// Mitsubishi GX Works2 project: BookEX2_3 Calculator   PLC: Q13UDV

// global labels: Global
VAR_GLOBAL
  bVar0 AT M5000 : BOOL;
  abArray0 AT M5010 : ARRAY [0..49] OF BOOL;
  sStr0 AT D5000 : STRING[199];
  sStr1 AT D5100 : STRING[199];
  sStr2 AT D5200 : STRING[199];
  sStr3 AT D5300 : STRING[199];
  sStr4 AT D5400 : STRING[199];
  sStr5 AT D5500 : STRING[199];
  sStr6 AT D5600 : STRING[199];
  sStr7 AT D5700 : STRING[199];
  sStr8 AT D5800 : STRING[199];
  sStr9 AT D5900 : STRING[199];
  iVar0 AT D4500 : INT;
  iVar1 AT D4501 : INT;
  iVar2 AT D4502 : INT;
  iVar3 AT D4503 : INT;
  iVar4 AT D4504 : INT;
  iVar5 AT D4505 : INT;
  iVar6 AT D4506 : INT;
  iVar7 AT D4507 : INT;
  iVar8 AT D4508 : INT;
  iVar9 AT D4509 : INT;
  dVar0 AT D4510 : DINT;
  dVar1 AT D4512 : DINT;
  dVar2 AT D4514 : DINT;
  dVar3 AT D4516 : DINT;
  dVar4 AT D4518 : DINT;
  dVar5 AT D4520 : DINT;
  dVar6 AT D4522 : DINT;
  dVar7 AT D4524 : DINT;
  dVar8 AT D4526 : DINT;
  dVar9 AT D4528 : DINT;
  wVar0 AT D4530 : WORD;
  wVar1 AT D4531 : WORD;
  wVar2 AT D4532 : WORD;
  wVar3 AT D4533 : WORD;
  wVar4 AT D4534 : WORD;
  wVar5 AT D4535 : WORD;
  wVar6 AT D4536 : WORD;
  wVar7 AT D4537 : WORD;
  wVar8 AT D4538 : WORD;
  wVar9 AT D4539 : WORD;
  dwVar0 AT D4540 : DWORD;
  dwVar1 AT D4542 : DWORD;
  dwVar2 AT D4544 : DWORD;
  dwVar3 AT D4546 : DWORD;
  dwVar4 AT D4548 : DWORD;
  dwVar5 AT D4550 : DWORD;
  dwVar6 AT D4552 : DWORD;
  dwVar7 AT D4554 : DWORD;
  dwVar8 AT D4556 : DWORD;
  dwVar9 AT D4558 : DWORD;
  fsVar0 AT D4560 : REAL;
  fsVar1 AT D4562 : REAL;
  fsVar2 AT D4564 : REAL;
  fsVar3 AT D4566 : REAL;
  fsVar4 AT D4568 : REAL;
  fsVar5 AT D4570 : REAL;
  fsVar6 AT D4572 : REAL;
  fsVar7 AT D4574 : REAL;
  fsVar8 AT D4576 : REAL;
  fsVar9 AT D4578 : REAL;
  fdVar0 AT D4580 : LREAL;
  tTime0 AT D4620 : TIME;
  tTime1 AT D4622 : TIME;
  tTime2 AT D4624 : TIME;
  tTime3 AT D4626 : TIME;
  tTime4 AT D4628 : TIME;
  tTime5 AT D4630 : TIME;
  tTime6 AT D4632 : TIME;
  tTime7 AT D4634 : TIME;
  tTime8 AT D4636 : TIME;
  tTime9 AT D4638 : TIME;
  tTime10 AT D4640 : TIME;
  bVar1 AT M5001 : BOOL;
  bVar2 AT M5002 : BOOL;
  bVar3 AT M5003 : BOOL;
  bVar4 AT M5004 : BOOL;
  bVar5 AT M5005 : BOOL;
  bVar6 AT M5006 : BOOL;
  bVar7 AT M5007 : BOOL;
  bVar8 AT M5008 : BOOL;
  bVar9 AT M5009 : BOOL;
  abArray1 AT M5060 : ARRAY [0..49] OF BOOL;
  abArray2 AT M5110 : ARRAY [0..49] OF BOOL;
  abArray3 AT M5160 : ARRAY [0..49] OF BOOL;
  abArray4 AT M5210 : ARRAY [0..49] OF BOOL;
  abArray5 AT M5260 : ARRAY [0..49] OF BOOL;
  abArray6 AT M5310 : ARRAY [0..49] OF BOOL;
  abArray7 AT M5360 : ARRAY [0..49] OF BOOL;
  abArray8 AT M5410 : ARRAY [0..49] OF BOOL;
  abArray9 AT M5460 : ARRAY [0..49] OF BOOL;
  fdVar1 AT D4584 : LREAL;
  fdVar2 AT D4588 : LREAL;
  fdVar3 AT D4592 : LREAL;
  fdVar4 AT D4596 : LREAL;
  fdVar5 AT D4600 : LREAL;
  fdVar6 AT D4604 : LREAL;
  fdVar7 AT D4608 : LREAL;
  fdVar8 AT D4612 : LREAL;
  fdVar9 AT D4616 : LREAL;
END_VAR
// user libraries (not included): HMI

FUNCTION_BLOCK Calculator
VAR_IN_OUT
  i_Key : INT;
END_VAR
VAR_OUTPUT
  fs_Val : REAL;
END_VAR
VAR
  fsValue1 : REAL;  (* 지난 입력숫자 *)
  fsValue2 : REAL;  (* 현재 표시숫자 *)
  iOperation : INT;
  fsDecimal : REAL;
  fsSign : REAL;
END_VAR
(* Key입력에 따른 처리*)
IF i_Key < 20 THEN
	CASE i_Key OF
		0..9 : 	IF fsDecimal = 0.0 THEN 		
					fsValue2 := (fsValue2 * 10.0) + INT_TO_REAL(i_Key);
				ELSE
					fsValue2 := fsValue2 + (fsDecimal * INT_TO_REAL(i_Key));
					fsDecimal := fsDecimal * 0.1;
				END_IF;
		11 : fsValue2 := fsValue2 * -1.0;
		12 : fsDecimal := 0.1;
		13 : fsDecimal := 0.0;
				fsValue2 := 0.0;
		14..17 : iOperation := i_Key;		
				fsValue1 := fsValue2;		
				fsValue2 := 0.0;
				fsDecimal := 0.0;
		10 : (* For equal-key input *)
				CASE iOperation OF
					14 :		fsValue2 := fsValue1 + fsValue2; 		
					15 : 		fsValue2 := fsValue1 - fsValue2;			
					16 : 		fsValue2 := fsValue1 * fsValue2;		
					17 : 		IF fsValue2 = 0.0 THEN  					
									fsValue2 := fsValue1;	
								ELSE
									fsValue2 := fsValue1 / fsValue2;
								END_IF;
				END_CASE;
				fsValue1 := fsValue2;		
				iOperation := 0; 
				fsDecimal := 0.0;
			ELSE
				i_Key := 99;	
	END_CASE;
	i_Key := 99;	
	fs_Val := fsValue2;
END_IF;
END_FUNCTION_BLOCK

PROGRAM SmallCalc
VAR
  Calculator_1 : Calculator;
END_VAR
(* structured ladder/FBD written out as ST: instructions are called as NAME(EN, inputs, outputs); _pN, _eN, _tN stand for wires *)
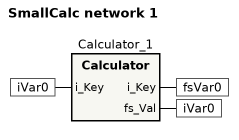
(* network 1 *)
Calculator_1(i_Key := iVar0, fs_Val => iVar0);
fsVar0 := Calculator_1.i_Key;
END_PROGRAM

PROGRAM ExSEG16
VAR
  aiClock : ARRAY [0..6] OF INT;
  aiMin : ARRAY [0..1] OF INT;
  aiSec : ARRAY [0..1] OF INT;
END_VAR
(* structured ladder/FBD written out as ST: instructions are called as NAME(EN, inputs, outputs); _pN, _eN, _tN stand for wires *)
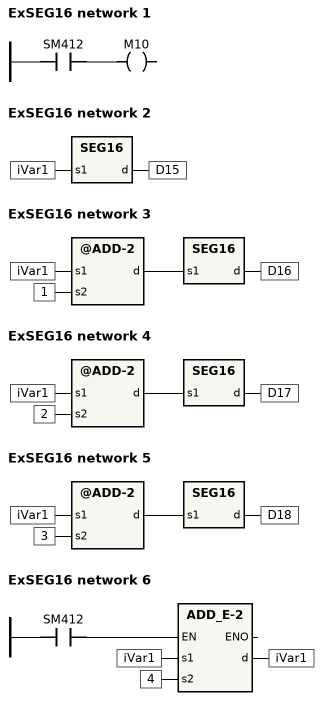
(* network 1 *)
M10 := SM412;
(* network 2 *)
D15 := SEG16(iVar1);
(* network 3 *)
D16 := SEG16(@ADD-2(iVar1, 1));
(* network 4 *)
D17 := SEG16(@ADD-2(iVar1, 2));
(* network 5 *)
D18 := SEG16(@ADD-2(iVar1, 3));
(* network 6 *)
ADD_E(SM412, iVar1, 4, iVar1);
END_PROGRAM

PROGRAM ExSEG7
VAR
  aiClock : ARRAY [0..6] OF INT;
  aiMin : ARRAY [0..1] OF INT;
  aiSec : ARRAY [0..1] OF INT;
END_VAR
(* structured ladder/FBD written out as ST: instructions are called as NAME(EN, inputs, outputs); _pN, _eN, _tN stand for wires *)
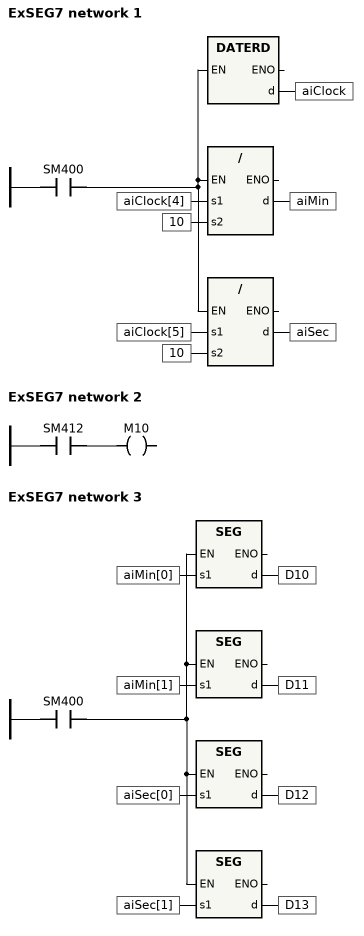
(* network 1 *)
DATERD(SM400, aiClock);
/(SM400, aiClock[4], 10, aiMin);
/(SM400, aiClock[5], 10, aiSec);
(* network 2 *)
M10 := SM412;
(* network 3 *)
SEG(SM400, aiMin[0], D10);
SEG(SM400, aiMin[1], D11);
SEG(SM400, aiSec[0], D12);
SEG(SM400, aiSec[1], D13);
END_PROGRAM

FUNCTION SEG16
VAR_INPUT
  i_Data : INT;
END_VAR
VAR
  Temp : WORD;
END_VAR
;
CASE i_Data MOD 16 OF
	0 :	Temp := H90FF;
	1 :	Temp := H100C;
	2 :	Temp := H0377;
	3 :	Temp := H023F;
	4 :	Temp := H038C;
	5 :	Temp := H03BB;
	6 :	Temp := H03FB;
	7 :	Temp := H000F;
	8 :	Temp := H03FF;
	9 :	Temp := H03BF;
	10 :	Temp := H03CF;
	11 :	Temp := H4A3F;
	12 :	Temp := H00F3;
	13 :	Temp := H483F;
	14 :	Temp := H01F3;
	15 :	Temp := H01C3;
END_CASE;
SEG16 := Temp;
END_FUNCTION
